SYSTEM TEST_SYS2 (* System Configuration for testing TEST_RES2 *)
  (* Standard: 61499-1 *)
  (* Version 0.0, 2004-06-08, JHC, Rockwell Automation *)
  APPLICATION APP1
  END_APPLICATION
  DEVICE DEV1 : FRAME_DEVICE
    RESOURCE INPUTS : PANEL_RESOURCE
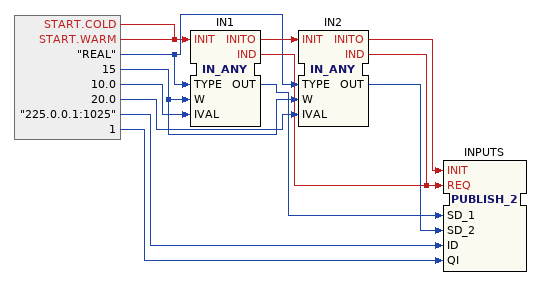
      FBS
        IN1 : IN_ANY;
        IN2 : IN_ANY;
        INPUTS : PUBLISH_2;
      END_FBS
      EVENT_CONNECTIONS
        START.COLD TO IN1.INIT;
        START.WARM TO IN1.INIT;
        IN1.INITO TO IN2.INIT;
        IN2.INITO TO INPUTS.INIT;
        IN1.IND TO INPUTS.REQ;
        IN2.IND TO INPUTS.REQ;
      END_CONNECTIONS
      DATA_CONNECTIONS
        IN1.OUT TO INPUTS.SD_1;
        IN2.OUT TO INPUTS.SD_2;
        "REAL" TO IN1.TYPE;
        "REAL" TO IN2.TYPE;
        15 TO IN1.W;
        15 TO IN2.W;
        10.0 TO IN1.IVAL;
        20.0 TO IN2.IVAL;
        "225.0.0.1:1025" TO INPUTS.ID;
        1 TO INPUTS.QI;
      END_CONNECTIONS
    END_RESOURCE
    RESOURCE TESTED : TEST_RES2
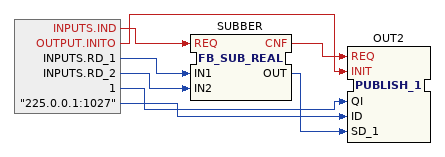
      FBS
        SUBBER : FB_SUB_REAL;
        OUT2 : PUBLISH_1;
      END_FBS
      EVENT_CONNECTIONS
        INPUTS.IND TO SUBBER.REQ;
        SUBBER.CNF TO OUT2.REQ;
        OUTPUT.INITO TO OUT2.INIT;
      END_CONNECTIONS
      DATA_CONNECTIONS
        INPUTS.RD_1 TO SUBBER.IN1;
        INPUTS.RD_2 TO SUBBER.IN2;
        1 TO OUT2.QI;
        "225.0.0.1:1027" TO OUT2.ID;
        SUBBER.OUT TO OUT2.SD_1;
      END_CONNECTIONS
    END_RESOURCE
    RESOURCE OUTPUTS : PANEL_RESOURCE
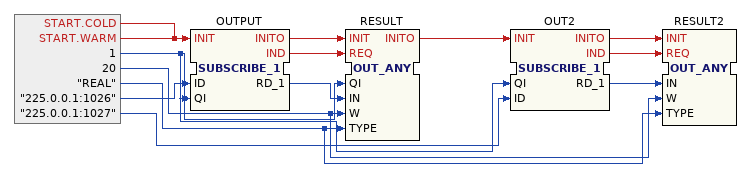
      FBS
        OUTPUT : SUBSCRIBE_1;
        RESULT : OUT_ANY;
        OUT2 : SUBSCRIBE_1;
        RESULT2 : OUT_ANY;
      END_FBS
      EVENT_CONNECTIONS
        START.COLD TO OUTPUT.INIT;
        START.WARM TO OUTPUT.INIT;
        OUTPUT.INITO TO RESULT.INIT;
        OUTPUT.IND TO RESULT.REQ;
        RESULT.INITO TO OUT2.INIT;
        OUT2.INITO TO RESULT2.INIT;
        OUT2.IND TO RESULT2.REQ;
      END_CONNECTIONS
      DATA_CONNECTIONS
        1 TO RESULT.QI;
        OUTPUT.RD_1 TO RESULT.IN;
        20 TO RESULT.W;
        "REAL" TO RESULT.TYPE;
        "225.0.0.1:1026" TO OUTPUT.ID;
        1 TO OUTPUT.QI;
        1 TO OUT2.QI;
        "225.0.0.1:1027" TO OUT2.ID;
        OUT2.RD_1 TO RESULT2.IN;
        20 TO RESULT2.W;
        "REAL" TO RESULT2.TYPE;
      END_CONNECTIONS
    END_RESOURCE
    DATA_CONNECTIONS
      "225.0.0.1:1025" TO TESTED.INPUT_ID;
      "225.0.0.1:1026" TO TESTED.OUTPUT_ID;
    END_CONNECTIONS
  END_DEVICE
  DATA_CONNECTIONS (* parameter values *)
    [2,1] TO DEV1.GRID;
    [100,100,150,150] TO DEV1.BOUNDS;
  END_CONNECTIONS
END_SYSTEM
